// TIA Portal V18 export
TYPE "SafetyGateUDT"
   STRUCT
      CMD : Struct
         RequestPB : Bool;   // 安全门请求按钮
      END_STRUCT;
      Status : Struct
         "Lock/Unlock Indicator" : Bool;   // 安全门锁定输出状态指示
         "INT" : Int;   // 安全门状态:1:已锁定,2:已解锁,3:安全门被打开
         Locked : Bool;   // 安全门已锁定
         Unlocked : Bool;   // 安全门已解锁
         Opened : Bool;   // 安全门已打开
      END_STRUCT;
   END_STRUCT;
END_TYPE
